TYPE ST_DataGridStationConfig :
STRUCT
	bEnabled : BOOL := FALSE; // To Enable Stations
	nActiveTestSteps	: UINT := 1;
	nActiveAteqDevices	: UINT := 1;
	nActiveValveBanks	: UINT := 1;
END_STRUCT
END_TYPE

(* stored: Version 1.1.0.1
   DUT ST_DataGridStationConfig: Id {bad48431-a915-0160-1460-5a36995f5fa3} *)
